// Mitsubishi GX Works2 project: 0715쉬프트   PLC: Q02/Q02H

PROGRAM MAIN
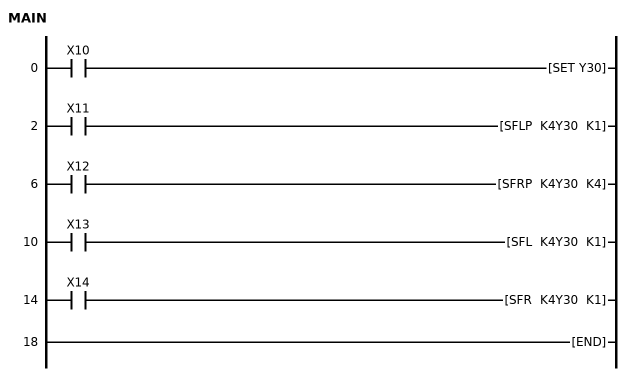
0     LD      X10
      SET     Y30
2     LD      X11
      SFLP    K4Y30 K1
6     LD      X12
      SFRP    K4Y30 K4
10    LD      X13
      SFL     K4Y30 K1
14    LD      X14
      SFR     K4Y30 K1
18    END
END_PROGRAM
